{attribute 'analysis' := '-33'}
TYPE MonitorTest :
STRUCT
    MonitorBeforeConnectDoesNotMatter			: BOOL;	
    SubscriptionsWillAllTriggerOnUpdateAsync	: BOOL;
    RegisterUnregisterIO						: BOOL;
    
    RegisterUnregisterMultipleIO1				: BOOL;
    RegisterUnregisterMultipleIO2				: BOOL;
    RegisterUnregisterMultipleIO3				: BOOL;
    RegisterUnregisterMultipleIO4				: BOOL;
    RegisterUnregisterMultipleIO5				: BOOL;
    RegisterUnregisterMultipleIO6				: BOOL;
    RegisterUnregisterMultipleIO7				: BOOL;
    RegisterUnregisterMultipleIO8				: BOOL;
    
    SubscribeIOUpdatesWhenValueChanges			: BOOL;
    SubscriptionsPersistReconnects				: BOOL;
    SubscribeIOShouldTriggerOnSubscribe			: BOOL;
    
    CanSubscribeToAllPlcTypes					: MonitorTestData;
END_STRUCT
END_TYPE

(* stored: Version 1.1.0.1
   DUT MonitorTest: Id {1fc35e25-4ef3-4a65-ae98-97be52d7f9ba} *)
